TYPE MyStruct :
STRUCT
	myInt: INT := 1;
	myBool: BOOL := FALSE;	
END_STRUCT
END_TYPE

(* stored: Version 1.1.0.1, ProductVersion 3.1.4018.9
   DUT MyStruct: Id {c28b6c7d-d444-4eb6-af9d-46f58c06b94a} *)
